{attribute addProperty BoxType "EJ1914-0000-0017"}
{attribute addProperty Id "FSOEAT %I*FSOE_4B534C96486"}
{attribute addProperty CRC "2308680718"}
{attribute addProperty SizeInBites "48"}
{attribute addProperty SizeInBytes "6"}
TYPE FSoE_Inputs_899BAC0E :
STRUCT
	{attribute addProperty Name "FSOE"}
	FSOE AT %I* : FSOE_4B534C96;
END_STRUCT
END_TYPE

(* stored: Version 1.2.0.0, ProductVersion 3.1.4024.9
   DUT FSoE_Inputs_899BAC0E: Id {217bb607-48b7-4d6b-91c2-11c20acc95d9} *)
